// TIA Portal V19 export
FUNCTION "PG Sim" : Void   // FC300, STL
{ S7_Optimized_Access := 'TRUE' }
// stored: AutoNumber false
BEGIN

NETWORK
TITLE = True = Process Valve is open.
      A     "ItemStatus".Y0904.Auto;
      =     "Y0904S";
      AN    "ItemStatus".Y0904.Auto;
      =     "Y0904R";

      A     "ItemStatus".Y0905.Auto;
      =     "Y0905S";
      AN    "ItemStatus".Y0905.Auto;
      =     "Y0905R";

      A     "ItemStatus".Y0906.Auto;
      =     "Y0906S";
      AN    "ItemStatus".Y0906.Auto;
      =     "Y0906R";

      A     "ItemStatus".Y0907.Auto;
      =     "Y0907S";
      AN    "ItemStatus".Y0907.Auto;
      =     "Y0907R";

      A     "ItemStatus".Y0908.Auto;
      =     "Y0908S";
      AN    "ItemStatus".Y0908.Auto;
      =     "Y0908R";

      A     "ItemStatus".Y0909.Auto;
      =     "Y0909S";
      AN    "ItemStatus".Y0909.Auto;
      =     "Y0909R";

      A     "ItemStatus".Y0910.Auto;
      =     "Y0910S";
      AN    "ItemStatus".Y0910.Auto;
      =     "Y0910R";

      A     "ItemStatus".Y0911.Auto;
      =     "Y0911S";
      AN    "ItemStatus".Y0911.Auto;
      =     "Y0911R";

      A     "ItemStatus".Y0912.Auto;
      =     "Y0912S";
      AN    "ItemStatus".Y0912.Auto;
      =     "Y0912R";


      A     "PG_Devices".V0552.IN.Activate;
      =     "ItemInfoScada".Items[68].Set_FB;
      AN    "PG_Devices".V0552.IN.Activate;
      =     "ItemInfoScada".Items[68].Reset_FB;

      A     "PG_Devices".V0934.IN.Activate;
      =     "ItemInfoScada".Items[69].Set_FB;
      AN    "PG_Devices".V0934.IN.Activate;
      =     "ItemInfoScada".Items[69].Reset_FB;

      A     "PG_Devices".V0935.IN.Activate;
      =     "ItemInfoScada".Items[70].Set_FB;
      AN    "PG_Devices".V0935.IN.Activate;
      =     "ItemInfoScada".Items[70].Reset_FB;

      A     "PG_Devices".V0936.IN.SV_1;
      =     "ItemInfoScada".Items[85].Set_FB;
      AN    "PG_Devices".V0936.IN.SV_1;
      =     "ItemInfoScada".Items[85].Reset_FB;

      A     "PG_Devices".V0940.IN.SV_1;
      =     "ItemInfoScada".Items[71].Set_FB;
      AN    "PG_Devices".V0940.IN.SV_1;
      =     "ItemInfoScada".Items[71].Reset_FB;


      A     "PG_Devices".V0941.IN.SV_1;
      =     "ItemInfoScada".Items[72].Set_FB;
      AN    "PG_Devices".V0941.IN.SV_1;
      =     "ItemInfoScada".Items[72].Reset_FB;


      A     "PG_Devices".V0942.IN.SV_1;
      =     "ItemInfoScada".Items[73].Set_FB;
      AN    "PG_Devices".V0942.IN.SV_1;
      =     "ItemInfoScada".Items[73].Reset_FB;


      A     "PG_Devices".V0943.IN.SV_1;
      =     "ItemInfoScada".Items[74].Set_FB;
      AN    "PG_Devices".V0943.IN.SV_1;
      =     "ItemInfoScada".Items[74].Reset_FB;

      A     "PG_Devices".V0944.IN.SV_1;
      =     "ItemInfoScada".Items[75].Set_FB;
      AN    "PG_Devices".V0944.IN.SV_1;
      =     "ItemInfoScada".Items[75].Reset_FB;

      A     "PG_Devices".V0945_SV1;
      =     "ItemInfoScada".Items[76].Set_FB;
      AN    "PG_Devices".V0945_SV1;
      =     "ItemInfoScada".Items[76].Reset_FB;

      A     "PG_Devices".V1021.IN_SV_1;
      =     "ItemInfoScada".Items[78].Set_FB;
      AN    "PG_Devices".V1021.IN_SV_1;
      =     "ItemInfoScada".Items[78].Reset_FB;

      A     "PG_Devices".V1023.IN.SV_1;
      =     "ItemInfoScada".Items[79].Set_FB;
      AN    "PG_Devices".V1023.IN.SV_1;
      =     "ItemInfoScada".Items[79].Reset_FB;

      A     "PG_Devices".V1024.IN.Activate;
      =     "ItemInfoScada".Items[80].Set_FB;
      AN    "PG_Devices".V1024.IN.Activate;
      =     "ItemInfoScada".Items[80].Reset_FB;

      A     "PG_Devices".V1025.IN.SV_1;
      =     "ItemInfoScada".Items[81].Set_FB;
      AN    "PG_Devices".V1025.IN.SV_1;
      =     "ItemInfoScada".Items[81].Reset_FB;

      A     "PG_Devices".V1027.IN.SV_1;
      =     "ItemInfoScada".Items[82].Set_FB;
      AN    "PG_Devices".V1027.IN.SV_1;
      =     "ItemInfoScada".Items[82].Reset_FB;

      A     "PG_Devices".V1083.IN.SV_1;
      =     "ItemInfoScada".Items[83].Set_FB;
      AN    "PG_Devices".V1083.IN.SV_1;
      =     "ItemInfoScada".Items[83].Reset_FB;

      A     "ItemStatus".M0940.Auto;
      =     "ItemInfoScada".Items[77].Set_FB;
      AN    "ItemStatus".M0940.Auto;
      =     "ItemInfoScada".Items[77].Reset_FB;

      A     "ItemStatus".M0941.Auto;
      =     "PG_Devices".DI_100_010_X02_4;
      =     "ItemInfoScada".Items[84].Set_FB;
      AN    "ItemStatus".M0941.Auto;
      =     "ItemInfoScada".Items[84].Reset_FB;
END_FUNCTION
